// Mitsubishi GX Works2 project: m04   PLC: Q02/Q02H

PROGRAM MAIN
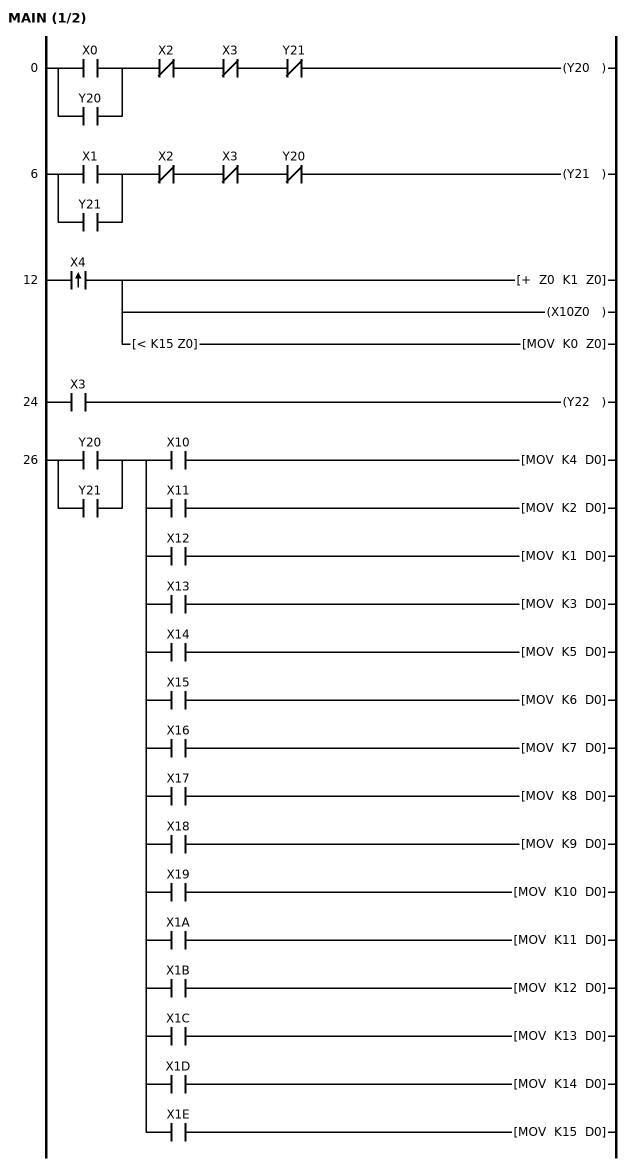
0     LD      X0
      OR      Y20
      ANI     X2
      ANI     X3
      ANI     Y21
      OUT     Y20
6     LD      X1
      OR      Y21
      ANI     X2
      ANI     X3
      ANI     Y20
      OUT     Y21
12    LDP     X4
      +       Z0 K1 Z0
      OUT     X10Z0
      AND<    K15 Z0
      MOV     K0 Z0
24    LD      X3
      OUT     Y22
26    LD      Y20
      OR      Y21
      MPS
      AND     X10
      MOV     K4 D0
      MRD
      AND     X11
      MOV     K2 D0
      MRD
      AND     X12
      MOV     K1 D0
      MRD
      AND     X13
      MOV     K3 D0
      MRD
      AND     X14
      MOV     K5 D0
      MRD
      AND     X15
      MOV     K6 D0
      MRD
      AND     X16
      MOV     K7 D0
      MRD
      AND     X17
      MOV     K8 D0
      MRD
      AND     X18
      MOV     K9 D0
      MRD
      AND     X19
      MOV     K10 D0
      MRD
      AND     X1A
      MOV     K11 D0
      MRD
      AND     X1B
      MOV     K12 D0
      MRD
      AND     X1C
      MOV     K13 D0
      MRD
      AND     X1D
      MOV     K14 D0
      MPP
      AND     X1E
      MOV     K15 D0
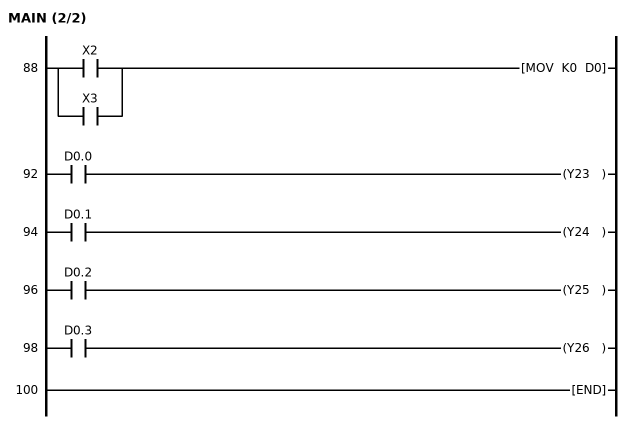
88    LD      X2
      OR      X3
      MOV     K0 D0
92    LD      D0.0
      OUT     Y23
94    LD      D0.1
      OUT     Y24
96    LD      D0.2
      OUT     Y25
98    LD      D0.3
      OUT     Y26
100   END
END_PROGRAM
